// Mitsubishi GX Works2 project: LRI - PLC - A1.Ã2   PLC: Q03UDV

PROGRAM MAIN
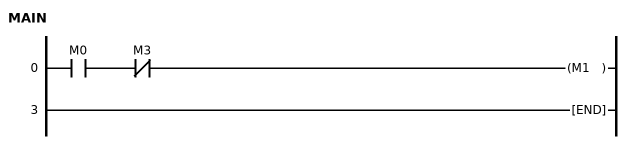
0     LD      M0
      ANI     M3
      OUT     M1
3     END
END_PROGRAM
